TYPE ST_ExtractiveControlValveParameters :
STRUCT
	timeToFullyOpenMs : DINT;
	calibrationTimeMs : DINT;
END_STRUCT
END_TYPE

(* stored: Version 1.1.0.1, ProductVersion 3.1.4024.9
   DUT ST_ExtractiveControlValveParameters: Id {02874832-6c8c-488c-848c-d0a9c2895470} *)
